// TIA Portal V17 export
// export: Created 2026-04-13T11:12:41.4655711Z, ExportSetting WithDefaults, DisplayName Totally Integrated Automation Portal, DisplayVersion V17 Update 4, DisplayName TIA Portal Openness, DisplayVersion V17 Update 4, DisplayName TIA Portal Version Control Interface, DisplayVersion V17, DisplayName SINAMICS Startdrive Advanced, DisplayVersion V17, DisplayName SINAMICS Startdrive G130, G150, S120, S150, SINAMICS MV, S210, DisplayVersion V17, DisplayName SINAMICS Startdrive G110M, G120, G120C, G120D, G120P, G115D, DisplayVersion V17, DisplayName STEP 7 Professional, DisplayVersion V17 Update 4, DisplayName STEP 7 Safety, DisplayVersion V17, DisplayName WinCC Professional, DisplayVersion V17 Update 4
FUNCTION_BLOCK "A3-脉冲轮询"   // FB12, SCL
{ S7_Optimized_Access := 'TRUE' }
VERSION : 0.1
// stored: AutoNumber true, IsIECCheckEnabled false, IsRetainMemResEnabled false, MemoryReserve 100, SetENOAutomatically false, UDAEnableTagReadback false
   VAR_INPUT
      num : Int;
      On_Time : Real;
   END_VAR
   VAR_OUTPUT
      output_1 : Bool;
      output_2 : Bool;
      output_3 : Bool;
      output_4 : Bool;
      output_5 : Bool;
      output_6 : Bool;
      output_7 : Bool;
      output_8 : Bool;
      output_9 : Bool;
      output_10 : Bool;
      output_11 : Bool;
      output_12 : Bool;
      output_13 : Bool;
      output_14 : Bool;
      output_15 : Bool;
      output_16 : Bool;
   END_VAR
   VAR_IN_OUT
      Stop_Time : Real;
      脉冲开关 : Bool;
      i : Int;
   END_VAR
   VAR
      t1 : TON_TIME;
      t2 { S7_SetPoint := 'True'} : TON_TIME;
      TM_FZ { ExternalAccessible := 'False'; ExternalVisible := 'False'; ExternalWritable := 'False'} : Bool;
      j : Int;
      output_ : Array[0..16] of Bool;
   END_VAR
   VAR RETAIN
      out_ : Array[0..16] of Bool;
   END_VAR
   VAR
      间隔时间 : Time := T#5s;
      运行时间 : Time := T#5s;
   END_VAR
   VAR_TEMP
      "m" : Int;
   END_VAR
BEGIN

   #间隔时间 := DINT_TO_TIME(REAL_TO_DINT(#Stop_Time * 1000.0));
   #运行时间 := DINT_TO_TIME(REAL_TO_DINT(#On_Time * 1000));


   #t1(IN := (1 <> #TM_FZ) AND #脉冲开关,
       PT := #间隔时间);

   #t2(IN := (1 = #TM_FZ) AND #脉冲开关,
       PT := #运行时间);

   IF #t1.Q THEN
       #TM_FZ := 1;
       #output_[#i] := 1;
   END_IF;

   IF #t2.Q THEN
       #TM_FZ := 0;
       #output_[#i] := 0;
       #i += 1;

   END_IF;

   IF #i >= #num OR #i < 0 OR (NOT #脉冲开关) THEN
       #i := 0;
       #TM_FZ := 0;
       FOR #j := 0 TO #num DO
           #output_[#j] := 0;
           IF (#j >= #num)
           THEN
               EXIT;
           END_IF;
       END_FOR;
   END_IF;


   FOR #m := 0 TO 16 DO
       IF #output_[#m] = TRUE THEN
           #out_[#m] := TRUE;
       ELSE
           #out_[#m] := FALSE;
       END_IF;
   END_FOR;
   #output_1 := #out_[0];
   #output_2 := #out_[1];
   #output_3 := #out_[2];
   #output_4 := #out_[3];
   #output_5 := #out_[4];
   #output_6 := #out_[5];
   #output_7 := #out_[6];
   #output_8 := #out_[7];
   #output_9 := #out_[8];
   #output_10 := #out_[9];

   #output_11 := #out_[10];
   #output_12 := #out_[11];
   #output_13 := #out_[12];
   #output_14 := #out_[13];
   #output_15 := #out_[14];
   #output_16 := #out_[15];
END_FUNCTION_BLOCK
